ABB RobotStudio station: ProyectoRemasterizado.rsstn

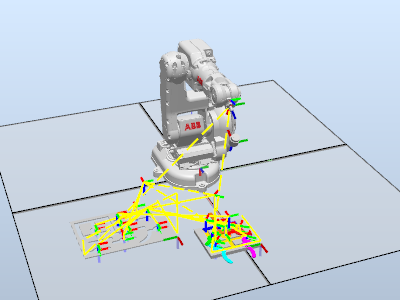
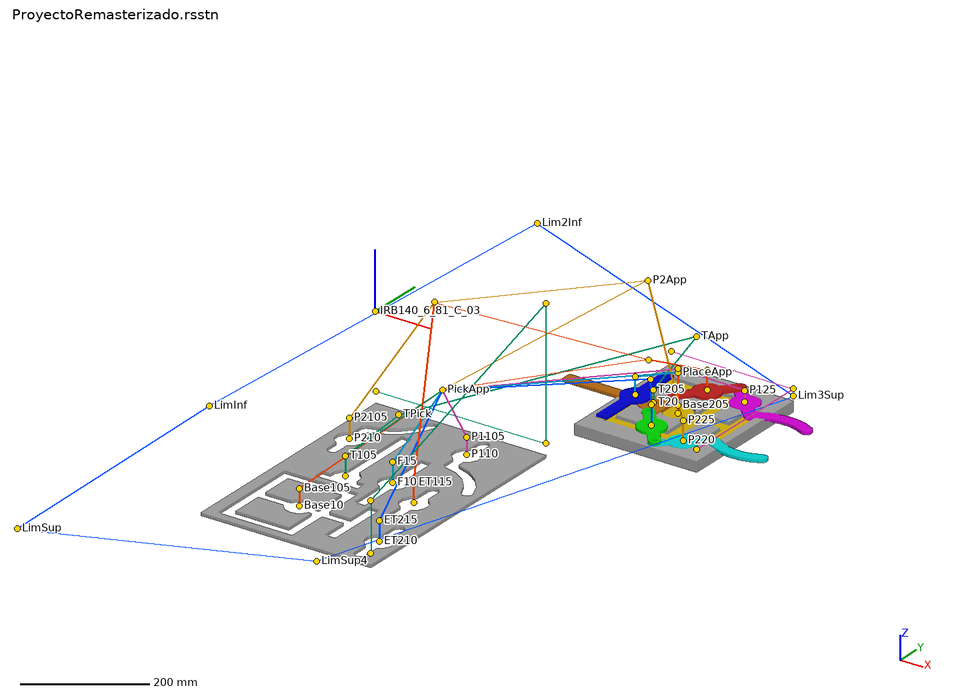
[picture v1: parts stored in the station drawn from their meshes, with robot base, taught points and paths (robot models come from the ABB library and are not in the file)]
Station ProyectoRemasterizado (saved by RobotStudio 22.2.9947.0)
Controller Proyecto2
  mechanical unit ROB_1: IRB140_6_81_C_03, 6 joints, base frame (0, 0, 0) mm
Layout (positions relative to the parent item):
  - IRB140_6_81_C_03 [mechanism, from Robots\IRB140_6_81_C_G_03.rslib] at (0, 0, 0) mm; joint values [0, 0, 0, 0, 0.5236, 0] (rad or m)
  - NewChupa [mechanism] at (506.29, 0, 679.5) mm, rotated rx 180 ry 60 rz 180 deg
      TCP Chupa at (-10.65, -116.78, 115.87) mm, rotated rx -90 ry 89.52 rz -179.52 deg
      links: Chupita2
  - PiezaACortarApoyoInicialV3_0 [part] at (541.15, -381.68, 0) mm, rotated rx 90 ry 0 rz 180 deg, size 320 x 5 x 470 mm
  - TablaDejarV3 [part] at (639.18, -60.56, -43.75) mm, rotated rx 90 ry 0 rz 180 deg, size 230 x 19 x 260 mm
  - BaseGripper [part] at (583.77, -50.6, 10) mm, rotated rx 90 ry 0 rz -180 deg, size 200 x 5 x 180 mm
  - EslabonTransmisor1 [part] at (606.72, 23.71, 20.75) mm, rotated rx 90 ry 0 rz -39.33 deg, size 50 x 5 x 124.5 mm
  - EslabonTransmisor2 [part] at (606.64, -124.82, 20.1) mm, rotated rx 90 ry 0 rz 40 deg, size 50 x 5 x 124.5 mm
  - Pinza1 [part] at (672.04, 32.31, 20) mm, rotated rx -90 ry 0 rz 45 deg, size 111 x 5 x 174 mm
  - Pinza2 [part] at (672.04, -133.51, 15.01) mm, rotated rx 90 ry 0 rz -45 deg, size 111 x 5 x 174 mm
  - PlacaRetencion [part] at (523.76, -50.61, 20) mm, rotated rx 90 ry 0 rz 0 deg, size 49.7 x 5 x 180 mm
  - T [part] at (573.29, -50.6, 15) mm, rotated rx 90 ry 0 rz 180 deg, size 190 x 5 x 80 mm
  - posB [smart component, from Components\Positioner.rslib]
      properties: Object=BaseGripper; Position=[0.28101 -0.63451 0]; Orientation=[1.5707963267949 0 3.14159265358979]; Reference=Global; ReferenceObject=(none)
  - posT [smart component, from Components\Positioner.rslib]
      properties: Object=T; Position=[0.29968 -0.52272 0]; Orientation=[1.5707963267949 0 1.5707963267949]; Reference=Global; ReferenceObject=(none)
  - posPR [smart component, from Components\Positioner.rslib]
      properties: Object=PlacaRetencion; Position=[0.37233 -0.48425 0]; Orientation=[1.5707963267949 0 0]; Reference=Global; ReferenceObject=(none)
  - posE1 [smart component, from Components\Positioner.rslib]
      properties: Object=EslabonTransmisor1; Position=[0.43971 -0.52448 0]; Orientation=[1.5707963267949 0 0]; Reference=Global; ReferenceObject=(none)
  - posE2 [smart component, from Components\Positioner.rslib]
      properties: Object=EslabonTransmisor2; Position=[0.47319 -0.6645 0]; Orientation=[1.5707963267949 0 0]; Reference=Global; ReferenceObject=(none)
  - posP1 [smart component, from Components\Positioner.rslib]
      properties: Object=Pinza1; Position=[0.40971 -0.3395 0.005]; Orientation=[-1.5707963267949 0 0]; Reference=Global; ReferenceObject=(none)
  - posP2 [smart component, from Components\Positioner.rslib]
      properties: Object=Pinza2; Position=[0.2292 -0.39631 0]; Orientation=[1.5707963267949 0 0]; Reference=Global; ReferenceObject=(none)
  - AttacherB [smart component, from Components\Attacher.rslib]
      properties: Parent=NewChupa; Flange=0; Child=BaseGripper; Mount=false; Offset=[0 0 0]; Orientation=[0 0 0]
  - DetacherB [smart component, from Components\Detacher.rslib]
      properties: Child=BaseGripper; KeepPosition=true
  - AttacherT [smart component, from Components\Attacher.rslib]
      properties: Parent=NewChupa; Flange=0; Child=T; Mount=false; Offset=[0 0 0]; Orientation=[0 0 0]
  - DetacherT [smart component, from Components\Detacher.rslib]
      properties: Child=T; KeepPosition=true
  - AttacherP1 [smart component, from Components\Attacher.rslib]
      properties: Parent=NewChupa; Flange=0; Child=Pinza1; Mount=false; Offset=[0 0 0]; Orientation=[0 0 0]
  - DetacherP1 [smart component, from Components\Detacher.rslib]
      properties: Child=Pinza1; KeepPosition=true
  - AttacherP2 [smart component, from Components\Attacher.rslib]
      properties: Parent=NewChupa; Flange=0; Child=Pinza2; Mount=false; Offset=[0 0 0]; Orientation=[0 0 0]
  - DetacherP2 [smart component, from Components\Detacher.rslib]
      properties: Child=Pinza2; KeepPosition=true
  - DetacherE1 [smart component, from Components\Detacher.rslib]
      properties: Child=EslabonTransmisor1; KeepPosition=true
  - AttacherE1 [smart component, from Components\Attacher.rslib]
      properties: Parent=NewChupa; Flange=0; Child=EslabonTransmisor1; Mount=false; Offset=[0 0 0]; Orientation=[0 0 0]
  - AttacherE2 [smart component, from Components\Attacher.rslib]
      properties: Parent=NewChupa; Flange=0; Child=EslabonTransmisor2; Mount=false; Offset=[0 0 0]; Orientation=[0 0 0]
  - DetacherE2 [smart component, from Components\Detacher.rslib]
      properties: Child=EslabonTransmisor2; KeepPosition=true
  - AttacherPR [smart component, from Components\Attacher.rslib]
      properties: Parent=NewChupa; Flange=0; Child=PlacaRetencion; Mount=false; Offset=[0 0 0]; Orientation=[0 0 0]
  - DetacherPR [smart component, from Components\Detacher.rslib]
      properties: Child=PlacaRetencion; KeepPosition=true
  - chupa [frame] at (127.2, 0.49, 126.37) mm, rotated rx -90 ry 89.52 rz -89.52 deg
Attachment: NewChupa is attached to IRB140_6_81_C_03 / Link6
Station signals: DI Home1, DI Home2, DI Home3, DI Home4, DI Home5, DI Home6, DI Home7
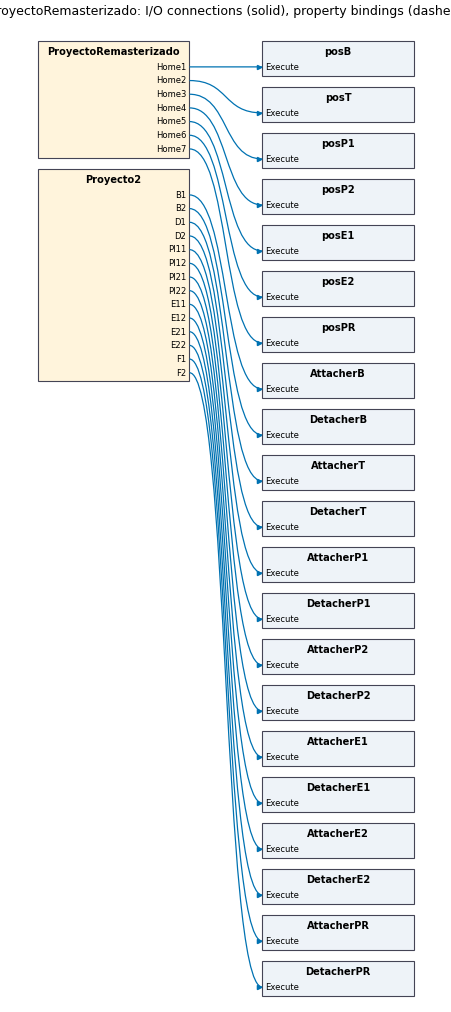
Station logic (signal -> signal, property => property):
  ProyectoRemasterizado.Home1 -> posB.Execute
  ProyectoRemasterizado.Home2 -> posT.Execute
  ProyectoRemasterizado.Home3 -> posP1.Execute
  ProyectoRemasterizado.Home4 -> posP2.Execute
  ProyectoRemasterizado.Home5 -> posE1.Execute
  ProyectoRemasterizado.Home6 -> posE2.Execute
  ProyectoRemasterizado.Home7 -> posPR.Execute
  Proyecto2.B1 -> AttacherB.Execute
  Proyecto2.B2 -> DetacherB.Execute
  Proyecto2.D1 -> AttacherT.Execute
  Proyecto2.D2 -> DetacherT.Execute
  Proyecto2.PI11 -> AttacherP1.Execute
  Proyecto2.PI12 -> DetacherP1.Execute
  Proyecto2.PI21 -> AttacherP2.Execute
  Proyecto2.PI22 -> DetacherP2.Execute
  Proyecto2.E11 -> AttacherE1.Execute
  Proyecto2.E12 -> DetacherE1.Execute
  Proyecto2.E21 -> AttacherE2.Execute
  Proyecto2.E22 -> DetacherE2.Execute
  Proyecto2.F1 -> AttacherPR.Execute
  Proyecto2.F2 -> DetacherPR.Execute
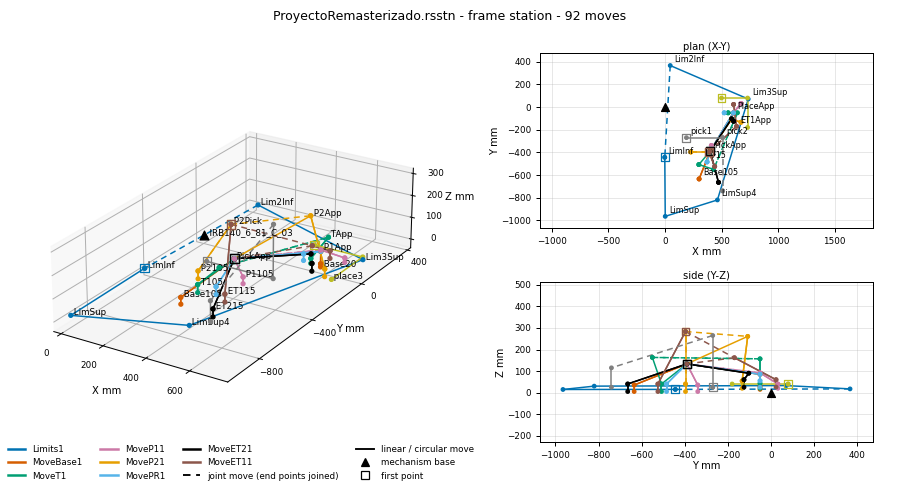
[picture p0: tool path of ProyectoRemasterizado.rsstn in frame station, 92 of 99 moves have a stored position in this frame; points joined in program order, loops and branches not executed]
Targets, tools, work objects and paths stored in the station, written as RAPID:
! task T_ROB1
MODULE CalibData
  PERS tooldata NewChupa:=[TRUE,[[127.2,0.485,126.368],[0.707106781,-0.005923775,0.707081968,0]],[1,[83.322,0.242,104.5],[1,0,0,0],0,0,0]];
  TASK PERS wobjdata World:=[FALSE,TRUE,"",[[0,0,0],[1,0,0,0]],[[0,0,0],[1,0,0,0]]];
  TASK PERS wobjdata NewPick:=[FALSE,TRUE,"",[[510,-270,5],[0,1,0,0]],[[0,0,0],[1,0,0,0]]];
  TASK PERS wobjdata NewPlace:=[FALSE,TRUE,"",[[730,80,20],[0,1,0,0]],[[0,0,0],[1,0,0,0]]];
ENDMODULE

! task T_ROB1
MODULE Module1
  CONST jointtarget Home:=[[0,0,0,0,30,0],[9E+09,9E+09,9E+09,9E+09,9E+09,9E+09]];
  CONST jointtarget Tool:=[[-89.3,42.5,-51.4,0,0,0],[9E+09,9E+09,9E+09,9E+09,9E+09,9E+09]];
  CONST robtarget LimInf:=[[-1.268558474,-443.594527115,14.946918722],[0,0.707106781,0.707106781,0],[-1,-2,1,0],[9E+09,9E+09,9E+09,9E+09,9E+09,9E+09]];
  CONST robtarget LimSup:=[[2.920655475,-964.874814922,14.510384672],[0,0.707106781,0.707106781,0],[-1,-2,1,0],[9E+09,9E+09,9E+09,9E+09,9E+09,9E+09]];
  CONST robtarget LimSup4:=[[463.722752628,-820,30.05181616],[0,0.707106781,0.707106781,0],[-1,-2,1,0],[9E+09,9E+09,9E+09,9E+09,9E+09,9E+09]];
  CONST robtarget Lim3Sup:=[[735.880314711,71.133179396,32.548470254],[-0.000000014,0.707106783,0.707106779,0.000000019],[0,-1,1,0],[9E+09,9E+09,9E+09,9E+09,9E+09,9E+09]];
  CONST robtarget Lim2Inf:=[[46.954799307,367.02539237,17.249386066],[0,0.707106781,0.707106781,0],[0,-1,1,0],[9E+09,9E+09,9E+09,9E+09,9E+09,9E+09]];
  CONST robtarget PickApp:=[[-110.342872773,120.113138802,-128.175841477],[0.707106781,0,0,-0.707106781],[-1,0,-1,1],[9E+09,9E+09,9E+09,9E+09,9E+09,9E+09]];
  CONST robtarget Base105:=[[-207.99,364.51,-30],[0.707106781,0,0,-0.707106781],[-1,0,-1,1],[9E+09,9E+09,9E+09,9E+09,9E+09,9E+09]];
  CONST robtarget Base10:=[[-207.99,364.511,0],[0.707106781,0,0,-0.707106781],[-1,0,-1,1],[9E+09,9E+09,9E+09,9E+09,9E+09,9E+09]];
  CONST robtarget PlaceApp:=[[-125.227,130.603,-65],[0.707106781,0,0,-0.707106781],[0,1,-1,1],[9E+09,9E+09,9E+09,9E+09,9E+09,9E+09]];
  CONST robtarget Base205:=[[-125.227,130.604,-8.971],[0.707106781,0,0,-0.707106781],[0,1,-1,1],[9E+09,9E+09,9E+09,9E+09,9E+09,9E+09]];
  CONST robtarget Base20:=[[-125.227,130.603,5],[0.707106781,0,0,-0.707106781],[0,1,-1,1],[9E+09,9E+09,9E+09,9E+09,9E+09,9E+09]];
  CONST robtarget T105:=[[-210.324,237.721,-35],[0.707106781,0,0,-0.707106781],[-1,0,-1,1],[9E+09,9E+09,9E+09,9E+09,9E+09,9E+09]];
  CONST robtarget T10:=[[-210.324,237.721,0],[0.707106781,0,0,-0.707106781],[-1,0,-1,1],[9E+09,9E+09,9E+09,9E+09,9E+09,9E+09]];
  CONST robtarget TPick:=[[-80.342872773,280.113138802,-158.175841477],[0.707106781,0,0,-0.707106781],[-1,0,-1,1],[9E+09,9E+09,9E+09,9E+09,9E+09,9E+09]];
  CONST robtarget TApp:=[[-90.227,130.604,-136.705],[0,0,0,1],[-1,-1,0,1],[9E+09,9E+09,9E+09,9E+09,9E+09,9E+09]];
  CONST robtarget T205:=[[-171.711,130.604,-22.457885204],[0,0,0,1],[-1,-1,-1,1],[9E+09,9E+09,9E+09,9E+09,9E+09,9E+09]];
  CONST robtarget T20:=[[-171.711,130.603,0],[0,0,0,1],[-1,-1,-1,1],[9E+09,9E+09,9E+09,9E+09,9E+09,9E+09]];
  CONST robtarget P1105:=[[-100.292,69.504,-30],[0.707106781,0,0,-0.707106781],[-1,0,-1,1],[9E+09,9E+09,9E+09,9E+09,9E+09,9E+09]];
  CONST robtarget P110:=[[-100.292,69.504,0],[0.707106781,0,0,-0.707106781],[-1,0,-1,1],[9E+09,9E+09,9E+09,9E+09,9E+09,9E+09]];
  CONST robtarget P1App:=[[-125.227,130.604,-71.705],[0.382683433,0,0,-0.923879532],[0,0,-1,1],[9E+09,9E+09,9E+09,9E+09,9E+09,9E+09]];
  CONST robtarget P125:=[[-57.955,47.693,-20],[0.382683433,0,0,-0.923879532],[0,0,-1,1],[9E+09,9E+09,9E+09,9E+09,9E+09,9E+09]];
  CONST robtarget P120:=[[-57.956,47.692,0],[0.382683432,0,0,-0.923879533],[0,0,-1,1],[9E+09,9E+09,9E+09,9E+09,9E+09,9E+09]];
  CONST robtarget P2Pick:=[[-121.178397921,126.307,-278.381942838],[0,0,0,1],[-1,1,-2,0],[9E+09,9E+09,9E+09,9E+09,9E+09,9E+09]];
  CONST robtarget P2105:=[[-280.797,126.307,-35],[0,0,0,1],[-1,1,-2,0],[9E+09,9E+09,9E+09,9E+09,9E+09,9E+09]];
  CONST robtarget P210:=[[-280.797,126.307,0],[0,0,0,1],[-1,1,-2,0],[9E+09,9E+09,9E+09,9E+09,9E+09,9E+09]];
  CONST robtarget P2App:=[[-142.214371526,187.704774603,-240.969916699],[0.382683433,0,0,-0.923879532],[0,0,-1,1],[9E+09,9E+09,9E+09,9E+09,9E+09,9E+09]];
  CONST robtarget P225:=[[-57.864,213.606,-34.204],[0.382683433,0,0,-0.923879532],[0,0,-1,1],[9E+09,9E+09,9E+09,9E+09,9E+09,9E+09]];
  CONST robtarget P220:=[[-57.956,213.515,0],[0.382683432,0,0,-0.923879533],[0,0,-1,1],[9E+09,9E+09,9E+09,9E+09,9E+09,9E+09]];
  CONST robtarget F15:=[[-137.666,214.247,-35],[0.707106781,0,0,-0.707106781],[-1,0,-1,1],[9E+09,9E+09,9E+09,9E+09,9E+09,9E+09]];
  CONST robtarget F10:=[[-137.666,214.247,0],[0.707106781,0,0,-0.707106781],[-1,0,-1,1],[9E+09,9E+09,9E+09,9E+09,9E+09,9E+09]];
  CONST robtarget F25:=[[-206.227,130.603,-35],[0.707106781,0,0,-0.707106781],[0,1,-1,1],[9E+09,9E+09,9E+09,9E+09,9E+09,9E+09]];
  CONST robtarget F20:=[[-206.231,130.606,-5],[0.707106781,0,0,-0.707106781],[0,1,-1,1],[9E+09,9E+09,9E+09,9E+09,9E+09,9E+09]];
  CONST robtarget ET215:=[[-36.814,394.504,-35],[0.707106781,0,0,-0.707106781],[-1,0,-1,1],[9E+09,9E+09,9E+09,9E+09,9E+09,9E+09]];
  CONST robtarget ET210:=[[-36.814,394.504,0],[0.707106781,0,0,-0.707106781],[-1,0,-1,1],[9E+09,9E+09,9E+09,9E+09,9E+09,9E+09]];
  CONST robtarget ET2App:=[[-141.14536065,182.779436275,-69.962726226],[0.382683433,0,0,-0.923879532],[0,0,-1,1],[9E+09,9E+09,9E+09,9E+09,9E+09,9E+09]];
  CONST robtarget ET225:=[[-123.166,204.988,-40],[0.422618262,0,0,-0.906307787],[0,0,-1,1],[9E+09,9E+09,9E+09,9E+09,9E+09,9E+09]];
  CONST robtarget ET220:=[[-123.36,204.828,-5.1],[0.422618262,0,0,-0.906307787],[0,0,-1,1],[9E+09,9E+09,9E+09,9E+09,9E+09,9E+09]];
  CONST robtarget ET115:=[[-70.294,254.478,-35],[0,0,0,1],[-1,1,-2,0],[9E+09,9E+09,9E+09,9E+09,9E+09,9E+09]];
  CONST robtarget ET110:=[[-70.293,254.479,0],[0,0,0,1],[-1,1,-2,0],[9E+09,9E+09,9E+09,9E+09,9E+09,9E+09]];
  CONST robtarget ET1App:=[[-97.458484126,249.43301943,-141.897823694],[0.336487213,0,0,-0.941688035],[-1,0,-1,1],[9E+09,9E+09,9E+09,9E+09,9E+09,9E+09]];
  CONST robtarget ET125:=[[-123.284,56.288,-40],[0.336487213,0,0,-0.941688035],[0,0,-1,1],[9E+09,9E+09,9E+09,9E+09,9E+09,9E+09]];
  CONST robtarget ET120:=[[-123.282,56.291,-5.75],[0.336487213,0,0,-0.941688035],[0,0,-1,1],[9E+09,9E+09,9E+09,9E+09,9E+09,9E+09]];
  CONST robtarget pick1:=[[190,-270,25],[0,0,1,0],[-2,1,1,0],[9E+09,9E+09,9E+09,9E+09,9E+09,9E+09]];
  CONST robtarget pick2:=[[510,-270,25],[0,0,1,0],[-1,1,2,0],[9E+09,9E+09,9E+09,9E+09,9E+09,9E+09]];
  CONST robtarget pick25:=[[510,-270,265],[0,0,1,0],[-1,1,2,0],[9E+09,9E+09,9E+09,9E+09,9E+09,9E+09]];
  CONST robtarget pick35:=[[510,-740,115],[0,0.707106781,0.707106781,0],[-1,-2,1,0],[9E+09,9E+09,9E+09,9E+09,9E+09,9E+09]];
  CONST robtarget pick3:=[[510,-740,25],[0,0.707106781,0.707106781,0],[-1,-2,1,0],[9E+09,9E+09,9E+09,9E+09,9E+09,9E+09]];
  CONST robtarget place1:=[[500,80,40],[0,0,1,0],[0,-2,-2,0],[9E+09,9E+09,9E+09,9E+09,9E+09,9E+09]];
  CONST robtarget place2:=[[730,80,40],[0,0,1,0],[0,-2,-3,0],[9E+09,9E+09,9E+09,9E+09,9E+09,9E+09]];
  CONST robtarget place3:=[[730,-180,40],[0,0,1,0],[-1,-3,-2,0],[9E+09,9E+09,9E+09,9E+09,9E+09,9E+09]];
  CONST jointtarget HomeFinal:=[[0,0,0,0,0,0],[9E+09,9E+09,9E+09,9E+09,9E+09,9E+09]];
  PROC main()
    Homing1;
    MoveBase1;
    MoveT1;
    MoveP11;
    MoveP21;
    MoveET11;
    MoveET21;
    MovePR1;
    Homing1;
  ENDPROC
  PROC Limits1()
    MoveJ LimInf,v150,fine,NewChupa\WObj:=wobj0;
    MoveL LimSup,v150,fine,NewChupa\WObj:=wobj0;
    MoveL LimSup4,v150,fine,NewChupa\WObj:=wobj0;
    MoveL Lim3Sup,v150,fine,NewChupa\WObj:=wobj0;
    MoveL Lim2Inf,v150,fine,NewChupa\WObj:=wobj0;
    MoveJ LimInf,v150,fine,NewChupa\WObj:=wobj0;
  ENDPROC
  PROC MoveBase1()
    MoveJ PickApp,v100,fine,NewChupa\WObj:=NewPick;
    MoveJ PickApp,v100,fine,NewChupa\WObj:=NewPick;
    MoveL Base105,v100,fine,NewChupa\WObj:=NewPick;
    MoveL Base10,v50,fine,NewChupa\WObj:=NewPick;
    Set B1;
    Set DO_01;
    WaitTime 0.5;
    MoveL Base105,v50,fine,NewChupa\WObj:=NewPick;
    MoveL PickApp,v100,fine,NewChupa\WObj:=NewPick;
    MoveL PlaceApp,v100,fine,NewChupa\WObj:=NewPlace;
    MoveL Base205,v100,fine,NewChupa\WObj:=NewPlace;
    MoveL Base20,v50,fine,NewChupa\WObj:=NewPlace;
    Reset DO_01;
    Set B2;
    WaitTime 0.5;
    MoveL Base205,v50,fine,NewChupa\WObj:=NewPlace;
    MoveL PlaceApp,v100,fine,NewChupa\WObj:=NewPlace;
    MoveL PickApp,v100,fine,NewChupa\WObj:=NewPick;
  ENDPROC
  PROC MoveT1()
    MoveL PickApp,v100,fine,NewChupa\WObj:=NewPick;
    MoveL T105,v100,fine,NewChupa\WObj:=NewPick;
    MoveL T10,v50,fine,NewChupa\WObj:=NewPick;
    Set D1;
    Set DO_01;
    WaitTime 0.5;
    MoveL T105,v100,fine,NewChupa\WObj:=NewPick;
    MoveL TPick,v100,fine,NewChupa\WObj:=NewPick;
    MoveJ TApp,v100,fine,NewChupa\WObj:=NewPlace;
    MoveL T205,v100,fine,NewChupa\WObj:=NewPlace;
    MoveL T20,v50,fine,NewChupa\WObj:=NewPlace;
    Set D2;
    Reset DO_01;
    WaitTime 0.5;
    WaitTime 0.5;
    MoveL T205,v100,fine,NewChupa\WObj:=NewPlace;
    MoveL TApp,v100,fine,NewChupa\WObj:=NewPlace;
    MoveJ TPick,v100,fine,NewChupa\WObj:=NewPick;
  ENDPROC
  PROC MoveP11()
    MoveL PickApp,v100,fine,NewChupa\WObj:=NewPick;
    MoveL P1105,v100,fine,NewChupa\WObj:=NewPick;
    MoveL P110,v50,fine,NewChupa\WObj:=NewPick;
    Set PI11;
    Set DO_01;
    WaitTime 0.5;
    MoveL P1105,v100,fine,NewChupa\WObj:=NewPick;
    MoveL PickApp,v100,fine,NewChupa\WObj:=NewPick;
    MoveJ P1App,v100,fine,NewChupa\WObj:=NewPlace;
    MoveL P125,v100,fine,NewChupa\WObj:=NewPlace;
    MoveL P120,v50,fine,NewChupa\WObj:=NewPlace;
    Set PI12;
    Reset DO_01;
    WaitTime 0.5;
    MoveL P125,v100,fine,NewChupa\WObj:=NewPlace;
    MoveL P1App,v100,fine,NewChupa\WObj:=NewPlace;
    MoveJ PickApp,v100,fine,NewChupa\WObj:=NewPick;
  ENDPROC
  PROC MoveP21()
    MoveJ P2Pick,v100,fine,NewChupa\WObj:=NewPick;
    MoveL P2105,v100,fine,NewChupa\WObj:=NewPick;
    MoveL P210,v50,fine,NewChupa\WObj:=NewPick;
    Set PI21;
    Set DO_01;
    WaitTime 0.5;
    MoveL P2105,v100,fine,NewChupa\WObj:=NewPick;
    MoveJ P2Pick,v100,fine,NewChupa\WObj:=NewPick;
    MoveJ P2App,v100,fine,NewChupa\WObj:=NewPlace;
    MoveL P225,v100,fine,NewChupa\WObj:=NewPlace;
    MoveL P220,v50,fine,NewChupa\WObj:=NewPlace;
    Set PI22;
    Reset DO_01;
    WaitTime 0.5;
    MoveL P225,v100,fine,NewChupa\WObj:=NewPlace;
    MoveL P2App,v100,fine,NewChupa\WObj:=NewPlace;
    MoveL PickApp,v100,fine,NewChupa\WObj:=NewPick;
  ENDPROC
  PROC MovePR1()
    MoveL PickApp,v100,fine,NewChupa\WObj:=NewPick;
    MoveL F15,v100,fine,NewChupa\WObj:=NewPick;
    MoveL F10,v50,fine,NewChupa\WObj:=NewPick;
    Set F1;
    Set DO_01;
    WaitTime 0.5;
    MoveL F15,v50,fine,NewChupa\WObj:=NewPick;
    MoveL PickApp,v100,fine,NewChupa\WObj:=NewPick;
    MoveL PlaceApp,v100,fine,NewChupa\WObj:=NewPlace;
    MoveL F25,v100,fine,NewChupa\WObj:=NewPlace;
    MoveL F20,v50,fine,NewChupa\WObj:=NewPlace;
    Reset DO_01;
    Set F2;
    WaitTime 0.5;
    MoveL F25,v50,fine,NewChupa\WObj:=NewPlace;
    MoveL PlaceApp,v100,fine,NewChupa\WObj:=NewPlace;
    MoveL PickApp,v100,fine,NewChupa\WObj:=NewPick;
  ENDPROC
  PROC MoveET21()
    MoveL PickApp,v100,fine,NewChupa\WObj:=NewPick;
    MoveL ET215,v100,fine,NewChupa\WObj:=NewPick;
    MoveL ET210,v50,fine,NewChupa\WObj:=NewPick;
    Set E21;
    Set DO_01;
    WaitTime 0.5;
    MoveL ET215,v50,fine,NewChupa\WObj:=NewPick;
    MoveL PickApp,v100,fine,NewChupa\WObj:=NewPick;
    MoveL ET2App,v100,fine,NewChupa\WObj:=NewPlace;
    MoveL ET225,v50,fine,NewChupa\WObj:=NewPlace;
    MoveL ET220,v50,fine,NewChupa\WObj:=NewPlace;
    WaitTime 0.5;
    Set E22;
    Reset DO_01;
    WaitTime 0.5;
    MoveL ET225,v50,fine,NewChupa\WObj:=NewPlace;
    MoveL ET2App,v100,fine,NewChupa\WObj:=NewPlace;
    MoveL PickApp,v100,fine,NewChupa\WObj:=NewPick;
  ENDPROC
  PROC MoveET11()
    MoveJ P2Pick,v100,fine,NewChupa\WObj:=NewPick;
    MoveL ET115,v100,fine,NewChupa\WObj:=NewPick;
    MoveL ET110,v50,fine,NewChupa\WObj:=NewPick;
    WaitTime 0.5;
    Set E11;
    Set DO_01;
    WaitTime 0.5;
    MoveL ET115,v100,fine,NewChupa\WObj:=NewPick;
    MoveL P2Pick,v100,fine,NewChupa\WObj:=NewPick;
    MoveJ ET1App,v100,fine,NewChupa\WObj:=NewPlace;
    MoveL ET125,v100,fine,NewChupa\WObj:=NewPlace;
    MoveL ET120,v50,fine,NewChupa\WObj:=NewPlace;
    WaitTime 0.5;
    Set E12;
    Reset DO_01;
    WaitTime 0.5;
    MoveL ET125,v100,fine,NewChupa\WObj:=NewPlace;
    MoveL ET1App,v100,fine,NewChupa\WObj:=NewPlace;
    MoveJ PickApp,v100,fine,NewChupa\WObj:=NewPick;
  ENDPROC
  PROC Homing1()
    MoveAbsJ Home,v200,fine,NewChupa\WObj:=NewPlace;
    Reset B1;
    Reset B2;
    Reset D1;
    Reset D2;
    Reset E11;
    Reset E12;
    Reset E21;
    Reset E22;
    Reset PI11;
    Reset PI12;
    Reset PI21;
    Reset PI22;
    Reset F1;
    Reset F2;
    Reset DO_01;
  ENDPROC
  PROC ToolSet1()
    MoveAbsJ Home,v300,fine,NewChupa\WObj:=wobj0;
    WaitDI DI_01,1;
    MoveAbsJ tool,v300,fine,NewChupa\WObj:=wobj0;
    WaitDI DI_01,1;
    MoveAbsJ Home,v300,fine,NewChupa\WObj:=wobj0;
  ENDPROC
  PROC DefinePick()
    MoveJ pick1,v300,fine,NewChupa\WObj:=World;
    WaitDI DI_01,1;
    MoveL pick2,v300,fine,NewChupa\WObj:=World;
    WaitDI DI_01,1;
    MoveL pick25,v300,fine,NewChupa\WObj:=World;
    MoveJ pick35,v300,fine,NewChupa\WObj:=World;
    MoveL pick3,v300,fine,NewChupa\WObj:=World;
    WaitDI DI_01,1;
    MoveAbsJ Home,v300,fine,NewChupa\WObj:=wobj0;
  ENDPROC
  PROC DefinePlace()
    MoveJ place1,v300,fine,NewChupa\WObj:=World;
    WaitDI DI_01,1;
    MoveL place2,v300,fine,NewChupa\WObj:=World;
    WaitDI DI_01,1;
    MoveL place3,v300,fine,NewChupa\WObj:=World;
    WaitDI DI_01,1;
    MoveAbsJ Home,v300,fine,NewChupa\WObj:=wobj0;
  ENDPROC
  PROC Final()
    MoveAbsJ HomeFinal,v300,fine,NewChupa\WObj:=NewPick;
    Reset DO_03;
  ENDPROC
ENDMODULE

